(* PLC project Unnamed, Unknown Unnamed 1 *)
(* stored: creationDateTime 2026-03-03T10:37:58, modificationDateTime 2026-03-03T12:51:17 *)

PROGRAM program0
  VAR
    START_PB : BOOL;
    MOTION_ENABLE : BOOL;
    STOP_PB : BOOL;
    FAULT_ACTIVE : BOOL;
    CYCLE_COMPLETE : BOOL;
    AUTO_RUN : BOOL;
    SR0 : SR;
  END_VAR

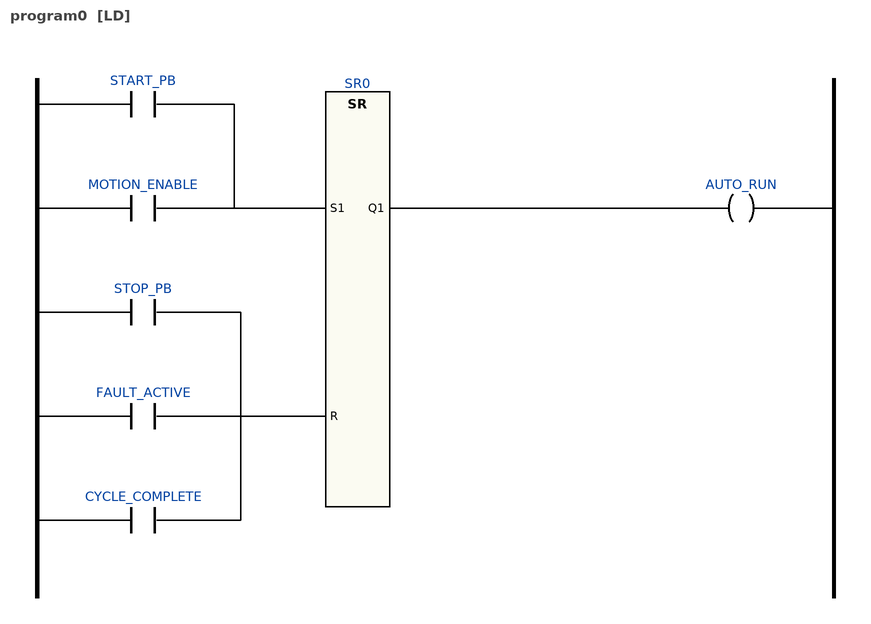
(* LD diagram, written out as Structured Text *)
SR0(S1 := START_PB OR MOTION_ENABLE, R := STOP_PB OR FAULT_ACTIVE OR CYCLE_COMPLETE);
AUTO_RUN := SR0.Q1;
END_PROGRAM

CONFIGURATION Config0
  RESOURCE Res0 ON PLC
    TASK task0(INTERVAL := T#20ms, PRIORITY := 0);
    PROGRAM instance0 WITH task0 : program0;
  END_RESOURCE
END_CONFIGURATION
